(* CODESYS project WagoAppDocker_Influx_v0.0.1.ecp

Project tree, tasks and I/O mapping:
  PFC200_G2_2ETH_RS_CAN_DPS : 750-8216 PFC200 PFC200 G2 2ETH RS CAN DPS, WAGO, order no. 0750-8216, version 5.13.2.22
    application Application
      libraries: ; SysProcess, 3.5.7.0 (System); WagoAppTime, 1.7.3.0 (WAGO)
      task PLC_Task (cyclic, interval t#50ms, priority 15) calls PLC_PRG
      program PLC_PRG [ST]
      Docker/
        data type typDockerPorts
        function block fbWagoAppDockerRun [ST]
        data type eRestartState
        data type typDockerVolume
      InfluxDb/
        function block WagoAppInfluxDb [ST]: CreateDatabase, Insert, Init, SWAP_BITS, GET_UTC
      program LOG_PRG [ST]
    Kbus : Kbus, WAGO, version 1.4.0.2
        unmapped channels: K-BUS diagnostics
      _8_DI_Generic : 075x-8DI, WAGO, order no. 075x-8DI, version 0.0.0.13
          settings: K-BUS Module slot index = 1
          unmapped channels: _IN
      _8_DO_Generic : 075x-8DO, WAGO, order no. 075x-8DO, version 0.0.0.13
          settings: K-BUS Module slot index = 2
          unmapped channels: _OUT
      _2AI_TC_K_Diagn : 0750-0469, WAGO, order no. 0750-0469, version 0.0.0.9
          settings: K-BUS Module slot index = 3
          input  iRawTc : INT  // _IINT 1
          unmapped channels: _IINT 2
    MODBUS
      MODBUS : MODBUS, WAGO, order no. n/a, version 1.1.1.15
    PROFIBUS
      PROFIBUS : PROFIBUS, WAGO, version 1.0.0.0 (disabled)
    CANbus
    Serial
      COM1 : COM1, WAGO, version 0.0.0.19
*)

// PFC200_G2_2ETH_RS_CAN_DPS/Application/Docker/typDockerPorts
TYPE typDockerPorts :
STRUCT
	wHostPort		: WORD;
	wContainerPort	: WORD;
END_STRUCT
END_TYPE

// PFC200_G2_2ETH_RS_CAN_DPS/Application/Docker/eRestartState
{attribute 'qualified_only'}
//{attribute 'strict'}
TYPE eRestartState :
(
	NO := 0,
	ON_FAILURE := 1,
	UNLESS_STOPPED := 2,
	ALWAYS := 3
);
END_TYPE

// PFC200_G2_2ETH_RS_CAN_DPS/Application/Docker/typDockerVolume
TYPE typDockerVolume :
STRUCT
	sLocalPath		: STRING;
	sContainerPath	: STRING;
END_STRUCT
END_TYPE

// PFC200_G2_2ETH_RS_CAN_DPS/Application/PLC_PRG
PROGRAM PLC_PRG
VAR
	xFirstScan					: BOOL := TRUE;
	tonOnDelay					: TON;
		
	fbDockerInflux				: fbWagoAppDockerRun;
	xDockerInfluxEn				: BOOL;
	xDockerInfluxIsRunning		: BOOL;
	sDockerInfluxContainerId	: STRING;
	eRestart 					: eRestartState := 2;
	xDockerInfluxError			: BOOL;
	xDockerInfluxWaiting		: BOOL;
	
	fbInfluxDb					: WagoAppInfluxDb;
	
	rTemperatureF		: REAL;
	rOldTemperatureF: REAL;
	diCreateDbResp: DINT;
	RTS_Resp: RTS_IEC_RESULT;
	sResponseString: STRING;
	
	sInfluxHostIp		: STRING := '10.6.10.238';
	sDatabaseName		: STRING := 'mydb';
	sDataObjName		: STRING := 'myvar';
	sFieldName			: STRING := 'myfield';
	
	tonLog				: TON;
	xLogData: BOOL;
	diLogResp: DINT;
	xDatabaseCreated: BOOL;

END_VAR

// run the docker container for the infux db
fbDockerInflux(
	xEnable:= xDockerInfluxEn,
	xBridgeHostNetwork := TRUE, 
	sImageName:= 'influxdb', 
	sContainerName:= 'influxpfc', 
	eRestartState:= eRestart, 
	xIsRunning=> xDockerInfluxIsRunning, 
	xError=> xDockerInfluxError,
	sContainerID=> sDockerInfluxContainerId);
	
	IF xFirstScan THEN
	xDockerInfluxEn := TRUE;
	// delay the db creation
	tonOnDelay(IN:= xDockerInfluxIsRunning, PT:= T#10S);
	IF tonOnDelay.Q THEN
		xFirstScan := FALSE;
	END_IF
END_IF
	
IF NOT xFirstScan AND NOT xDatabaseCreated THEN
	//diCreateDbResp := SysProcess.SysProcessExecuteCommand2('curl http://10.6.10.20:8086/query --data-urlencode $'q=CREATE DATABASE "myTemps"$'',sResponseString, 100, RTS_Resp);
	diCreateDbResp := fbInfluxDb.CreateDatabase(sInfluxHostIp, sDatabaseName);
	IF diCreateDbResp <> 0 THEN
		xDatabaseCreated := TRUE;
	END_IF
END_IF
	
rTemperatureF := (INT_TO_REAL(IoConfig_Globals_Mapping.iRawTc / 10) * 1.8) + 32;
tonLog(IN:= (xDatabaseCreated AND NOT xLogData), PT := T#1S);
IF  tonLog.Q THEN
	xLogData := TRUE;
END_IF
	
rOldTemperatureF := rTemperatureF;
	
IF xLogData THEN
	diLogResp := fbInfluxDb.Insert(sInfluxHostIp,sDatabaseName,sDataObjName,sFieldName, REAL_TO_STRING(rTemperatureF));
	IF diLogResp > 1 THEN
		xLogData := FALSE;
	END_IF
END_IF

END_PROGRAM

// PFC200_G2_2ETH_RS_CAN_DPS/Application/Docker/fbWagoAppDockerRun
FUNCTION_BLOCK fbWagoAppDockerRun
VAR_IN_OUT
	xEnable				: BOOL;
	aPorts				: ARRAY[*] OF WORD;
	aVolumes			: ARRAY[*] OF typDockerVolume;
END_VAR
VAR_INPUT
	sImageName			: STRING;
	sTag				: STRING := '';
	sContainerName		: STRING := '';
	xBridgeHostNetwork	: BOOL;
	eRestartState		: eRestartState;
END_VAR
VAR_OUTPUT
	xIsRunning			: BOOL;
	xError				: BOOL;
	xBusy				: BOOL;
	sContainerID		: STRING;
END_VAR
VAR
	rtInit					: R_TRIG;
	rtRun					: R_TRIG;
	rtGracefulClose			: R_TRIG;
	sDockerRunString		: STRING(255);
	sPortString				: STRING;
	ubPorts					: DINT;
	lbPorts					: DINT;
	i						: DINT;
	xDockerStringReady		: BOOL;
	diDockerRunResp			: DINT;
	sShellReturn			: STRING;
	pShellResult			: RTS_IEC_RESULT;
	xDockerRun				: BOOL;
	xStopContainer			: BOOL;
	sDockerStopCommand		: STRING(255);
	diStopCommandResp		: DINT;
	sStopCommandShellReturn	: STRING;
END_VAR

rtInit(CLK:= xEnable);
IF rtInit.Q THEN
	// show busy
	xDockerStringReady := FALSE;
	diDockerRunResp := 0;
	diStopCommandResp := 0;
	xError := FALSE;
	xBusy := TRUE;
	
	// initialize the string values
	sDockerRunString := 'docker run -d ';
	sPortString := '';
	
	CASE eRestartState OF
		0: sDockerRunString := CONCAT(sDockerRunString, '--restart no ');
		1: sDockerRunString := CONCAT(sDockerRunString, '--restart on-failure ');
		2: sDockerRunString := CONCAT(sDockerRunString, '--restart unless-stopped ');
		3: sDockerRunString := CONCAT(sDockerRunString, '--restart always ');
	END_CASE
	// format command for the ports
	ubPorts:=UPPER_BOUND (aPorts,1);
	lbPorts:=LOWER_BOUND (aPorts,1); 
	IF NOT xBridgeHostNetwork THEN
		IF ubPorts > 0 THEN
			FOR i := lbPorts TO ubPorts DO
				sPortString := CONCAT6(sPortString, '-p ',INT_TO_STRING(aPOrts[i]), ':', INT_TO_STRING(aPOrts[i]), ' ');
			END_FOR
		END_IF
	ELSIF xBridgeHostNetwork THEN
		sPortString := '--network=host ';
	END_IF
	sDockerRunString := CONCAT(sDockerRunString, sPortString);
	
	sDockerRunString := CONCAT(sDockerRunString, '-v /etc/localtime:/etc/localtime ');
	
	// check for name and add to call 
	IF sContainerName <> '' THEN
		sDockerRunString := CONCAT4(sDockerRunString, '--name ', sContainerName, ' ');
	END_IF
	sDockerRunString := CONCAT(sDockerRunString, sImageName);
	xDockerStringReady := TRUE;
END_IF

rtRun(CLK:= xDockerStringReady AND xEnable);
IF rtRun.Q THEN
	xDockerRun := TRUE;
END_IF

IF xDockerRun THEN
	diDockerRunResp := SysProcess.SysProcessExecuteCommand2(pszCommand:= sDockerRunString, pszStdOut:= sShellReturn, udiStdOutLen:= 10, pResult:= pShellResult);
	IF diDockerRunResp = 1 THEN
		xError := TRUE;
		xDockerRun := FALSE;
	ELSIF diDockerRunResp > 0 THEN
		sContainerID := sShellReturn;
		xIsRunning := TRUE;
		xDockerRun := FALSE;
	END_IF
END_IF

// close the container
rtGracefulClose(CLK:= xIsRunning AND NOT xEnable);
IF rtGracefulClose.Q THEN
	diStopCommandResp := 0;
	xError := FALSE;
	xStopContainer := TRUE;
END_IF

IF xStopContainer THEN
	sDockerStopCommand := CONCAT('docker rm -f ', sContainerID);
	diStopCommandResp := SysProcess.SysProcessExecuteCommand2(pszCommand:= sDockerStopCommand, pszStdOut:= sStopCommandShellReturn, udiStdOutLen:= 10, pResult:= pShellResult);
	IF diStopCommandResp = 1 THEN
		xError := TRUE;
		xStopContainer := FALSE;
	ELSIF diStopCommandResp > 0 THEN
		sContainerID := sShellReturn;
		xIsRunning := FALSE;
		xStopContainer := FALSE;
	END_IF
END_IF

END_FUNCTION_BLOCK

// PFC200_G2_2ETH_RS_CAN_DPS/Application/InfluxDb/WagoAppInfluxDb
FUNCTION_BLOCK WagoAppInfluxDb
VAR_INPUT
END_VAR
VAR_OUTPUT
END_VAR
VAR
	//sHostIp	: STRING;
	sInsertString	: STRING(255);
END_VAR

METHOD CreateDatabase : DINT
VAR_INPUT
	sHostIp			: STRING;
	sDatabaseName	: STRING;
END_VAR
VAR
	sHoldString		: STRING(255);
	myResult		: RTS_IEC_RESULT;
	sResponse		: STRING;
END_VAR
CreateDatabase := 0;

//sHoldString := 'curl http://10.6.10.20:8086/query --data-urlencode $'q=CREATE DATABASE "myTemps"$'';
sHoldString := CONCAT5('curl http://', sHostIp,':8086/query --data-urlencode $'q=CREATE DATABASE "',sDatabaseName,'"$'');

CreateDatabase := SysProcess.SysProcessExecuteCommand2(sHoldString, sResponse, 100, myResult);
END_METHOD

METHOD Insert : DINT
VAR_INPUT
	sHostIp			: STRING;
	sDatabaseName	: STRING;
	sObjectName		: STRING;
	sFieldName		: STRING;
	sFieldValue		: STRING;
END_VAR
VAR
	sHoldString		: STRING(255);
	diCurrentTime	: DWORD;
	myResult: RTS_IEC_RESULT;
	sResponse: STRING;
	ltCurrentTime: LTIME;
	sUTC: STRING;
END_VAR

//curl -i -XPOST 'http://localhost:8086/write?db=mydb' --data-binary 'cpu_load_short,host=server01,region=us-west value=0.64 1434055562000000000'
Insert := 0;

sUTC := GET_UTC();
//ltCurrentTime := FuGetLongTime();
//diCurrentTime := SWAP_BITS(LTIME_TO_DWORD(ltCurrentTime));

sHoldString := CONCAT7('curl -i -XPOST $'http://',sHostIp,':8086/write?db=', sDatabaseName, '$' --data-binary $'',sObjectName,',');
sHoldString := CONCAT8(sHoldString,'mytag=1 ',sFieldName, '=',sFieldValue,' ',sUTC, '$'');

sInsertString := sHoldString;

Insert := SysProcess.SysProcessExecuteCommand2(sHoldString,sResponse, 100, myResult);
END_METHOD

METHOD Init : DINT
VAR_INPUT
	sHost		: STRING;
END_VAR
sHostIp := sHost;
END_METHOD

METHOD SWAP_BITS : DWORD
VAR_INPUT
	dwIn	: DWORD;
END_VAR

VAR
	i		: INT;
	dwHold	: DWORD;
END_VAR
dwHold.0 := dwIn.31;
dwHold.1 := dwIn.30;
dwHold.2 := dwIn.29;
dwHold.3 := dwIn.28;
dwHold.4 := dwIn.27;
dwHold.5 := dwIn.26;
dwHold.6 := dwIn.25;
dwHold.7 := dwIn.24;
dwHold.8 := dwIn.23;
dwHold.9 := dwIn.22;
dwHold.10 := dwIn.21;
dwHold.11 := dwIn.20;
dwHold.12 := dwIn.19;
dwHold.13 := dwIn.18;
dwHold.14 := dwIn.17;
dwHold.15 := dwIn.16;
dwHold.16 := dwIn.15;
dwHold.17 := dwIn.14;
dwHold.18 := dwIn.13;
dwHold.19 := dwIn.12;
dwHold.20 := dwIn.11;
dwHold.21 := dwIn.10;
dwHold.22 := dwIn.9;
dwHold.23 := dwIn.8;
dwHold.24 := dwIn.7;
dwHold.25 := dwIn.6;
dwHold.26 := dwIn.5;
dwHold.27 := dwIn.4;
dwHold.28 := dwIn.3;
dwHold.29 := dwIn.2;
dwHold.30 := dwIn.1;
dwHold.31 := dwIn.0;

SWAP_BITS:=dwHold;
END_METHOD

METHOD GET_UTC : STRING
VAR_INPUT
END_VAR

VAR
	sUTC: STRING;
	myResult: RTS_IEC_RESULT;
END_VAR
SysProcess.SysProcessExecuteCommand2('date +%s', sUTC, 10,myResult);
GET_UTC := CONCAT(sUTC,'0000000000');
END_METHOD

END_FUNCTION_BLOCK

// PFC200_G2_2ETH_RS_CAN_DPS/Application/LOG_PRG
PROGRAM LOG_PRG
VAR
END_VAR

END_PROGRAM
